{attribute 'qualified_only'}
{attribute 'to_string'}
// Fault codes for FB_AnalogOutput. Range convention matches the shared
// device-fault convention (see docs/7-Architecture.md):
//   0        No fault
//   1-9      Timeouts
//   10-19    Feedback / hardware / signal
//   20-29    State violations
//   40-49    Configuration / process limits
//   50-59    Interlocks / permissives
TYPE E_AnalogOutput_Fault :
(
    None          := 0,

    BadQuality    := 10,    // inpQuality latched to BAD past cfgQualityFaultAfter
    ClampLow      := 11,    // commanded EU below cfgMinCv (raises when cfgClampAsFault)
    ClampHigh     := 12,    // commanded EU above cfgMaxCv (raises when cfgClampAsFault)

    BadConfig     := 40     // cfgRawMin > cfgRawMax, cfgEuMin >= cfgEuMax, etc.
);
END_TYPE

(* stored: Version 1.1.0.1, ProductVersion 3.1.4026.12
   DUT E_AnalogOutput_Fault: Id {a1100004-0004-0000-0000-000000000001} *)
